Yaskawa INFORM job: WRARC_.JBI

/JOB

//NAME WRARC

//INST

///DATE 2013/12/17 10:48

///ATTR SC,RW

///GROUP1 RB1

NOP

SET I003 0

JUMP *ARC_ON IF I004=1

ARCOF

JUMP *ARC_OFF

*ARC_ON

ARCON AC=I020 AV=IO21

*ARC_OFF

END
